FUNCTION F_Real_To_Byte : BYTE
VAR_INPUT
	nByte	: INT; //x (1 - 4) byte it get from real
	fReal	: REAL;	 
END_VAR
VAR
	nPos	: LWORD;
END_VAR


CASE nByte OF
	1:
		nPos := 0;
	2:
		nPos := 7;
	3:
		nPos := 14;
	4:
		nPos := 21;
ELSE
	RETURN;	
END_CASE

MEMCPY(ADR(F_Real_To_Byte),(ADR(fReal)+ nPos),8);

END_FUNCTION

(* stored: Version 1.1.0.1, ProductVersion 3.1.4024.11
   POU F_Real_To_Byte: Id {1c05a09a-6515-4f79-be97-dc34c63d765d}, SpecialFunc None *)
